FUNCTION_BLOCK XtsXPU
VAR
END_VAR

METHOD GetMoverInterface : BOOL
VAR_INPUT
END_VAR
END_METHOD

END_FUNCTION_BLOCK

(* stored: Version 1.1.0.1, ProductVersion 3.1.4024.12
   POU XtsXPU: Id {a76d70c0-85a8-4201-b7ed-df139d53b29f}, SpecialFunc None
   Method GetMoverInterface: Id {52f53c6d-8f9b-4420-aa70-9b69f63ace23} *)
